// TIA Portal V20 export
TYPE "typeSequenceControlNodeJobInterface"
// stored: Namespace Unit1.Em13
   STRUCT
      PICKJob2 : "LER_typeJobInterface";
      conveyorUnloadJob3 : "LER_typeJobInterface";
      stackNgBoxUnloadJob4 : "LER_typeJobInterface";
   END_STRUCT;
END_TYPE
